PROGRAM MAIN_prec_arch
VAR
	input : ARRAY[0..4] OF LREAL := [1,1,1,1,1];	
	out : ARRAY[0..0] OF LREAL;
	FB_NN : FB_Dense_v1;
	
	runtime_profiler : PROFILER;
	profiler_data : PROFILERSTRUCT;
	
	buf_idx : UINT := 0;
	profiler_buffer : ARRAY [0..1000] OF DWORD;
	
	MeasureFinished : BOOL := TRUE;

	

END_VAR


runtime_profiler(START := TRUE, RESET := TRUE);
FB_NN(pointer_input := ADR(input),pointer_output:= ADR(out));

runtime_profiler(START := FALSE);
profiler_data := runtime_profiler.DATA;

IF NOT MeasureFinished THEN
	profiler_buffer[buf_idx] := profiler_data.LastExecTime;
	buf_idx := buf_idx+1; 
	buf_idx := buf_idx MOD (SIZEOF(profiler_buffer)/SIZEOF(DWORD)); // len of profiler_buffer
END_IF
IF FB_NN.flag_AreWeightsLoaded THEN
	MeasureFinished := TRUE;
END_IF

END_PROGRAM

(* stored: Version 1.1.0.1, ProductVersion 3.1.4024.12
   POU MAIN_prec_arch: Id {af0fbab6-e2d8-454e-acb6-91e2fbecb631}, SpecialFunc None *)
